FUNCTION ImageHasCompatibleElementType : BOOL
VAR_INPUT
	Image : ITcVnImage;	
END_VAR
VAR_IN_OUT
	CompatibleElementTypes : ARRAY[*] OF ETcVnElementType;
END_VAR
VAR
	i : DINT;
END_VAR

IF NOT IsValidImage(Image) THEN
	RETURN;
END_IF

FOR i := LOWER_BOUND(CompatibleElementTypes, 1) TO UPPER_BOUND(CompatibleElementTypes, 1) DO
	IF ImageHasElementType(Image, CompatibleElementTypes[i]) THEN
		ImageHasCompatibleElementType := TRUE;
		RETURN;
	END_IF
END_FOR

END_FUNCTION

(* stored: Version 1.1.0.1, ProductVersion 3.1.4024.13
   POU ImageHasCompatibleElementType: Id {324cdee2-5a01-4ee1-9221-770fdf0fa0b6}, SpecialFunc None *)
